PROGRAM BS02PL_LineBackground
VAR
END_VAR

MAIN.stLine_BS02PL.fbLine(stLine:=MAIN.stLine_BS02PL);
MAIN.stLine_BS02PL.stStation_BS02PL01.fbStation(
				stLine:=MAIN.stLine_BS02PL,
				stStation:=MAIN.stLine_BS02PL.stStation_BS02PL01);

END_PROGRAM

(* stored: Version 1.1.0.1, ProductVersion 3.1.4024.15
   POU BS02PL_LineBackground: Id {9c33aca0-62b3-4ad6-ba4a-f1844b291f32}, SpecialFunc None *)
